{attribute 'strict'}
TYPE E_VisuCtrlInitializingPopUpFrameSelector :
(
	VISU_CTRL_INITIALIZING_FRAME_E_STOP 					:= 0,
	VISU_CTRL_INITIALIZING_FRAME_DOOR_LOCK 					:= 1,	
	VISU_CTRL_INITIALIZING_FRAME_RESET_BUTTON				:= 3	
);
END_TYPE

(* stored: Version 1.1.0.1, ProductVersion 3.1.4024.9
   DUT E_VisuCtrlInitializingPopUpFrameSelector: Id {61aa58af-54e6-4683-819e-1dccb326328e} *)
